{attribute 'qualified_only'}
{attribute 'strict'}
{attribute 'to_string'}
TYPE EScreenSide :
(
	Unknown := 0,
    Back,
    Front
);
END_TYPE

(* stored: Version 1.1.0.1, ProductVersion 3.1.4024.12
   DUT EScreenSide: Id {4207e3f2-9acc-4f70-b73d-f942b95cab77} *)
